Yaskawa INFORM job: X2_7,1(-165,-90)0.JBI

/JOB
//NAME X2_7,1(-165,-90)0
//POS
///NPOS 176,176,176,10,0,0
///TOOL 0
///POSTYPE PULSE
///PULSE
C00000=-39612,-76551,-106625,19964,71626,76894
C00001=-136747,-74177,-105509,19364,71994,77223
C00002=-161484,-91945,-110261,14957,103238,71453
C00003=-134320,-92773,-58904,770,74516,77205
C00004=-134673,-92214,-54444,791,72061,77068
C00005=-134820,-91899,-52604,800,71092,77011
C00006=-134844,-90764,-50356,804,70293,76998
C00007=-134845,-90951,-50699,804,70408,76998
C00008=-134847,-90902,-50689,804,70426,76998
C00009=-135220,-93018,-51550,819,69873,76866
C00010=-134847,-90902,-50689,804,70426,76998
C00011=-134345,-91899,-57067,774,73834,77192
C00012=-131570,-88662,-77507,437,88211,78221
C00013=-134523,-105271,-82138,1688,77555,77123
C00014=-134783,-105110,-77920,1731,75048,76999
C00015=-134891,-104934,-76180,1749,74070,76947
C00016=-134915,-104095,-74155,1758,73257,76927
C00017=-134916,-104246,-74475,1757,73376,76929
C00018=-134967,-104172,-74385,1762,73360,76911
C00019=-135343,-106731,-75345,1806,72644,76769
C00020=-134967,-104172,-74385,1762,73360,76911
C00021=-134596,-104670,-80422,1700,76809,77088
C00022=-136142,-134585,-102052,6475,55790,75677
C00023=-135158,-114824,-94391,5988,60976,76349
C00024=-135004,-111643,-89125,6022,59367,76321
C00025=-134943,-110346,-86998,6037,58724,76309
C00026=-134968,-109685,-85073,6101,57885,76253
C00027=-134968,-109829,-85430,6091,58030,76261
C00028=-135015,-109667,-85346,6108,58065,76244
C00029=-135392,-112540,-86390,6315,57265,76048
C00030=-135015,-109667,-85346,6108,58065,76244
C00031=-135230,-114226,-92783,6055,60303,76285
C00032=-156325,-82511,-105508,20476,72304,69745
C00033=-137289,-84891,-120500,10173,76813,76449
C00034=-137303,-139323,-128947,10263,31295,76421
C00035=-31263,-162610,-128854,9653,11963,76756
C00036=11604,-169116,-125244,11553,23484,75880
C00037=126218,-114256,-117174,36511,17097,65041
C00038=160817,-140540,-109431,13437,75130,4571
C00039=171379,-93893,-58713,11798,67401,-77246
C00040=173134,-92396,-53907,11771,65008,-76852
C00041=173854,-91715,-51934,11761,64060,-76687
C00042=173992,-90510,-49657,11819,63274,-76718
C00043=173854,-91715,-51934,11761,64060,-76687
C00044=173987,-90681,-50014,11807,63403,-76706
C00045=175295,-92334,-50710,11680,62808,-76287
C00046=173987,-90681,-50014,11807,63403,-76706
C00047=173264,-91392,-52007,11815,64350,-76873
C00048=171504,-92964,-56866,11837,66737,-77269
C00049=148375,-121212,-86833,17149,72660,-74878
C00050=158259,-104656,-80103,12690,76821,-80970
C00051=159746,-104467,-75973,12677,74202,-80717
C00052=160359,-104277,-74268,12676,73177,-80607
C00053=160467,-103358,-72208,12716,72383,-80652
C00054=160359,-104277,-74268,12676,73177,-80607
C00055=160417,-103437,-72504,12711,72529,-80655
C00056=161432,-105657,-73351,12654,71766,-80373
C00057=160417,-103437,-72504,12711,72529,-80655
C00058=159802,-103665,-74229,12711,73547,-80766
C00059=158313,-103959,-78409,12718,76144,-81021
C00060=158569,-141300,-112815,9916,80451,-74883
C00061=158798,-111123,-96627,9897,85638,-81727
C00062=159864,-112561,-93144,9862,82666,-81595
C00063=160305,-112963,-91680,9854,81520,-81533
C00064=160413,-112330,-89778,9865,80674,-81563
C00065=160399,-112442,-90081,9863,80802,-81557
C00066=160441,-112453,-90085,9860,80794,-81544
C00067=161459,-115136,-91053,9809,79898,-81262
C00068=160441,-112453,-90085,9860,80794,-81544
C00069=159997,-112112,-91574,9867,81924,-81608
C00070=158926,-110847,-95124,9896,84850,-81745
C00071=160682,-88290,-103875,4722,98055,-77441
C00072=135323,-109589,-91807,-1190,81195,-77099
C00073=133148,-118247,-66270,-328,65792,-77561
C00074=133675,-116428,-61229,-353,63627,-77373
C00075=133898,-115629,-59169,-363,62770,-77293
C00076=133957,-114036,-56802,-368,62133,-77271
C00077=133948,-114328,-57228,-367,62244,-77274
C00078=133917,-114378,-57192,-366,62197,-77284
C00079=134431,-116412,-57765,-387,61506,-77104
C00080=133917,-114378,-57192,-366,62197,-77284
C00081=133693,-115200,-59270,-355,63052,-77365
C00082=133162,-117080,-64355,-330,65213,-77555
C00083=138392,-136781,-94069,-1907,68850,-75598
C00084=132958,-105241,-81767,-1134,77157,-77611
C00085=133235,-105027,-77525,-1173,74661,-77491
C00086=133288,-104357,-75613,-1183,73831,-77465
C00087=133388,-103974,-73743,-1199,72877,-77421
C00088=133382,-104139,-74110,-1197,73019,-77424
C00089=133359,-104157,-74082,-1195,72992,-77432
C00090=133697,-106715,-75039,-1234,72272,-77307
C00091=133359,-104157,-74082,-1195,72992,-77432
C00092=133244,-104394,-75853,-1178,73958,-77481
C00093=132967,-104722,-80150,-1137,76429,-77601
C00094=138196,-141776,-101555,-7752,51920,-74477
C00095=133428,-114968,-94090,-4986,60450,-76927
C00096=133334,-111722,-88803,-5027,58864,-76892
C00097=133296,-110401,-86667,-5046,58229,-76877
C00098=133336,-109716,-84733,-5107,57396,-76822
C00099=133330,-109844,-85063,-5097,57532,-76831
C00100=133345,-109829,-85035,-5104,57524,-76825
C00101=133683,-112700,-86073,-5289,56713,-76650
C00102=133345,-109829,-85035,-5104,57524,-76825
C00103=133382,-111175,-87184,-5084,58155,-76839
C00104=133477,-114487,-92506,-5041,59728,-76875
C00105=141752,-106189,-89524,-13947,62090,-73527
C00106=139337,-93830,-82897,-11067,68844,-75160
C00107=137529,-73575,-73827,-8033,82117,-76735
C00108=128276,-76076,-75002,-6276,80740,-79812
C00109=127910,-97020,-84121,-7469,66652,-79182
C00110=129021,-107399,-90499,-8627,61500,-78401
C00111=153189,-105013,-101528,-11669,72335,-68251
C00112=139010,-107606,-90936,13602,98517,-80019
C00113=140479,-111236,-88693,13669,95112,-79881
C00114=141104,-112370,-87439,13712,93689,-79820
C00115=153388,-106096,-85115,15113,93243,-75565
C00116=152633,-104764,-86492,15083,94863,-75632
C00117=150753,-101320,-88700,15024,98237,-75883
C00118=160913,-92989,-79235,24173,97682,-73194
C00119=151950,-102059,-74371,18707,88669,-80768
C00120=154021,-103736,-71350,18921,85616,-80507
C00121=156769,-103064,-69269,19190,84099,-79774
C00122=166959,-95557,-66660,19849,83821,-76203
C00123=165303,-95872,-68594,19733,85187,-76570
C00124=162983,-94318,-71559,19573,88219,-76909
C00125=177330,-95873,-81273,-5233,90327,-76206
C00126=140937,-97211,-77708,-6493,80278,-75430
C00127=139211,-88421,-70354,-5139,84673,-76249
C00128=139768,-88806,-68107,-5161,83133,-75995
C00129=129086,-91534,-69174,-4923,81722,-79583
C00130=127811,-91239,-71468,-4873,83202,-80077
C00131=128888,-101422,-79212,-5537,77745,-79462
C00132=137877,-110952,-72155,-1851,88703,-77001
C00133=139734,-110509,-58972,-1399,80627,-76317
C00134=140249,-110783,-54995,-1319,78047,-76125
C00135=142549,-109961,-52712,-916,77094,-75392
C00136=133855,-111346,-52444,-6859,76619,-78478
C00137=133337,-111815,-54560,-7332,77679,-78736
C00138=134028,-111541,-58531,-7151,80301,-78669
C00139=164216,-109032,-67322,9813,79557,-67843
C00140=178281,-110359,-72151,20782,77591,-61941
C00141=158557,-96763,-53299,19671,77500,-80212
C00142=161145,-96732,-49400,20091,74655,-79786
C00143=163160,-95939,-47445,20342,73441,-79290
C00144=171236,-91338,-45159,23204,70710,-76469
C00145=169251,-92133,-47198,23012,72018,-76926
C00146=166209,-92508,-51159,22625,74900,-77459
C00147=149807,-144247,-110382,14568,75746,-63630
C00148=126218,-114256,-117174,36511,17097,65041
C00149=118793,-153239,-128782,32477,23422,65112
C00150=11604,-169116,-125244,11553,23484,75880
C00151=-137287,-84892,-120500,10191,64594,76446
C00152=-160620,-101266,-113002,23179,68693,67515
C00153=-142986,-103863,-89383,14232,64402,73407
C00154=-140772,-93459,-83022,11808,69469,74770
C00155=-137440,-81398,-77271,8908,76967,76533
C00156=-127109,-84097,-78453,6470,75327,80029
C00157=-129407,-96992,-84444,8303,67122,78735
C00158=-131023,-111117,-91294,10327,58712,77443
C00159=-137851,-122869,-93518,6619,76408,76346
C00160=-142777,-98750,-78529,7299,79569,74803
C00161=-140556,-88306,-70608,5557,85156,75864
C00162=-139393,-89232,-68583,5550,83361,76182
C00163=-128741,-91750,-69554,5331,81947,79756
C00164=-129199,-91422,-71906,5329,83587,79669
C00165=-130949,-106780,-81238,6593,74219,78605
C00166=-147304,-112155,-77948,4789,93136,74966
C00167=-140707,-86501,-53635,6284,90799,77049
C00168=-140521,-88167,-50612,6312,88084,76975
C00169=-139464,-88632,-48933,6512,86739,77253
C00170=-126799,-90769,-49711,8803,84964,81310
C00171=-127817,-90605,-51563,8619,86280,81066
C00172=-128613,-89112,-54690,8476,89025,80988
C00173=-161484,-91945,-110261,14957,103238,71453
C00174=-136747,-74177,-105509,19364,71994,77223
C00175=-39612,-76551,-106625,19964,71626,76894
BC00000=295325,674563,1075175
BC00001=353535,895977,1075175
BC00002=353535,975867,1075175
BC00003=346138,1016365,1074941
BC00004=346138,1016365,1074941
BC00005=346138,1016365,1074941
BC00006=346138,1016365,1074941
BC00007=346138,1016365,1074941
BC00008=346138,1016365,1074941
BC00009=346138,1016365,1074941
BC00010=346138,1016365,1074941
BC00011=346138,1016365,1074941
BC00012=345633,1015596,1047596
BC00013=345436,1039539,1075175
BC00014=345436,1039539,1075175
BC00015=345436,1039539,1075175
BC00016=345436,1039539,1075175
BC00017=345436,1039539,1075175
BC00018=345436,1039539,1075175
BC00019=345436,1039539,1075175
BC00020=345436,1039539,1075175
BC00021=345436,1039539,1075175
BC00022=345633,1030850,1075175
BC00023=346084,1031619,1075175
BC00024=346084,1031619,1075175
BC00025=346084,1031619,1075175
BC00026=346084,1031619,1075175
BC00027=346084,1031619,1075175
BC00028=346084,1031619,1075175
BC00029=346084,1031619,1075175
BC00030=346084,1031619,1075175
BC00031=346084,1031619,1075175
BC00032=381896,966588,1075175
BC00033=353816,923989,1075175
BC00034=353816,923989,1075175
BC00035=379773,1126391,1075175
BC00036=335955,1030285,1075175
BC00037=312632,1138057,1075175
BC00038=340753,1115300,1075175
BC00039=317618,1085268,1067802
BC00040=317618,1085268,1067802
BC00041=317618,1085268,1067802
BC00042=317618,1085268,1067802
BC00043=317618,1085268,1067802
BC00044=317618,1085268,1067802
BC00045=317618,1085268,1067802
BC00046=317618,1085268,1067802
BC00047=317618,1085268,1067802
BC00048=317618,1085268,1067802
BC00049=304558,1071386,1075175
BC00050=304527,1061353,1075175
BC00051=304527,1061353,1075175
BC00052=304527,1061353,1075175
BC00053=304527,1061353,1075175
BC00054=304527,1061353,1075175
BC00055=304527,1061353,1075175
BC00056=304527,1061353,1075175
BC00057=304527,1061353,1075175
BC00058=304527,1061353,1075175
BC00059=304527,1061353,1075175
BC00060=297809,1030861,1075175
BC00061=297809,1030861,1075175
BC00062=297809,1030861,1075175
BC00063=297809,1030861,1075175
BC00064=297809,1030861,1075175
BC00065=297809,1030861,1075175
BC00066=297809,1030861,1075175
BC00067=297809,1030861,1075175
BC00068=297809,1030861,1075175
BC00069=297809,1030861,1075175
BC00070=297809,1030861,1075175
BC00071=323405,1100688,1075175
BC00072=345633,1145987,1075175
BC00073=341431,1080783,1075175
BC00074=341431,1080783,1075175
BC00075=341431,1080783,1075175
BC00076=341431,1080783,1075175
BC00077=341431,1080783,1075175
BC00078=341431,1080783,1075175
BC00079=341431,1080783,1075175
BC00080=341431,1080783,1075175
BC00081=341431,1080783,1075175
BC00082=341431,1080783,1075175
BC00083=345633,1085057,1075175
BC00084=345596,1084288,1075175
BC00085=345596,1084288,1075175
BC00086=345596,1084288,1075175
BC00087=345596,1084288,1075175
BC00088=345596,1084288,1075175
BC00089=345596,1084288,1075175
BC00090=345596,1084288,1075175
BC00091=345596,1084288,1075175
BC00092=345596,1084288,1075175
BC00093=345596,1084288,1075175
BC00094=345633,1092894,1075175
BC00095=345573,1092125,1075175
BC00096=345573,1092125,1075175
BC00097=345573,1092125,1075175
BC00098=345573,1092125,1075175
BC00099=345573,1092125,1075175
BC00100=345573,1092125,1075175
BC00101=345573,1092125,1075175
BC00102=345573,1092125,1075175
BC00103=345573,1092125,1075175
BC00104=345573,1092125,1075175
BC00105=338421,1101651,1075175
BC00106=338421,1101651,1075175
BC00107=338421,1101651,1075175
BC00108=338421,1101651,1075175
BC00109=338421,1101651,1075175
BC00110=338421,1101651,1075175
BC00111=329561,1092894,1075175
BC00112=285121,1016140,1075175
BC00113=285121,1016140,1075175
BC00114=285121,1016140,1075175
BC00115=285121,1016140,1075175
BC00116=285121,1016140,1075175
BC00117=285121,1016140,1075175
BC00118=322883,1030260,1075175
BC00119=305317,1037338,1075175
BC00120=305317,1037338,1075175
BC00121=305317,1037338,1075175
BC00122=305317,1037338,1075175
BC00123=305317,1037338,1075175
BC00124=305317,1037338,1075175
BC00125=352461,1065435,1075175
BC00126=338520,1089250,1075175
BC00127=338520,1089250,1075175
BC00128=338520,1089250,1075175
BC00129=338520,1089250,1075175
BC00130=338520,1089250,1075175
BC00131=338520,1089250,1075175
BC00132=329561,1063988,1075175
BC00133=329824,1054944,1075175
BC00134=329824,1054944,1075175
BC00135=329824,1054944,1075175
BC00136=329824,1054944,1075175
BC00137=329824,1054944,1075175
BC00138=329824,1054944,1075175
BC00139=331300,1058024,1069499
BC00140=329561,1042367,1075175
BC00141=308437,1059196,1075175
BC00142=308437,1059196,1075175
BC00143=308437,1059196,1075175
BC00144=308437,1059196,1075175
BC00145=308437,1059196,1075175
BC00146=308437,1059196,1075175
BC00147=340753,1115300,1075175
BC00148=312632,1138057,1075175
BC00149=312632,1138057,1075175
BC00150=335955,1030285,1075175
BC00151=353817,923990,1075175
BC00152=381896,966588,1075175
BC00153=338906,1022094,1075175
BC00154=338906,1022094,1075175
BC00155=338906,1022094,1075175
BC00156=338906,1022094,1075175
BC00157=338906,1022094,1075175
BC00158=338906,1022094,1075175
BC00159=330026,1050278,1075175
BC00160=338884,1034595,1075175
BC00161=338884,1034595,1075175
BC00162=338884,1034595,1075175
BC00163=338884,1034595,1075175
BC00164=338884,1034595,1075175
BC00165=338884,1034595,1075175
BC00166=330026,1059203,1075175
BC00167=326517,1040873,1058771
BC00168=326517,1040873,1058771
BC00169=326517,1040873,1058771
BC00170=326517,1040873,1058771
BC00171=326517,1040873,1058771
BC00172=326517,1040873,1058771
BC00173=353535,975867,1075175
BC00174=353535,895977,1075175
BC00175=295325,674563,1075175
EC00000=-1463287,-556475
EC00001=-1463287,-556475
EC00002=-1463287,-556475
EC00003=-1463287,-556475
EC00004=-1463287,-556475
EC00005=-1463287,-556475
EC00006=-1463287,-556475
EC00007=-1463287,-556475
EC00008=-1463287,-556475
EC00009=-1463287,-556475
EC00010=-1463287,-556475
EC00011=-1463287,-556475
EC00012=-1463287,-556475
EC00013=-1463287,-556475
EC00014=-1463287,-556475
EC00015=-1463287,-556475
EC00016=-1463287,-556475
EC00017=-1463287,-556475
EC00018=-1463287,-556475
EC00019=-1463287,-556475
EC00020=-1463287,-556475
EC00021=-1463287,-556475
EC00022=-1463287,-556475
EC00023=-1463287,-556475
EC00024=-1463287,-556475
EC00025=-1463287,-556475
EC00026=-1463287,-556475
EC00027=-1463287,-556475
EC00028=-1463287,-556475
EC00029=-1463287,-556475
EC00030=-1463287,-556475
EC00031=-1463287,-556475
EC00032=-1463287,-556475
EC00033=-1463287,-556475
EC00034=-1463287,-556475
EC00035=-1463287,-556475
EC00036=-1595090,-3837
EC00037=-1729339,556475
EC00038=-1729339,556475
EC00039=-1729339,556475
EC00040=-1729339,556475
EC00041=-1729339,556475
EC00042=-1729339,556475
EC00043=-1729339,556475
EC00044=-1729339,556475
EC00045=-1729339,556475
EC00046=-1729339,556475
EC00047=-1729339,556475
EC00048=-1729339,556475
EC00049=-1729339,556475
EC00050=-1729339,556475
EC00051=-1729339,556475
EC00052=-1729339,556475
EC00053=-1729339,556475
EC00054=-1729339,556475
EC00055=-1729339,556475
EC00056=-1729339,556475
EC00057=-1729339,556475
EC00058=-1729339,556475
EC00059=-1729339,556475
EC00060=-1729339,556475
EC00061=-1729339,556475
EC00062=-1729339,556475
EC00063=-1729339,556475
EC00064=-1729339,556475
EC00065=-1729339,556475
EC00066=-1729339,556475
EC00067=-1729339,556475
EC00068=-1729339,556475
EC00069=-1729339,556475
EC00070=-1729339,556475
EC00071=-1729339,556475
EC00072=-1729339,556475
EC00073=-1729339,556475
EC00074=-1729339,556475
EC00075=-1729339,556475
EC00076=-1729339,556475
EC00077=-1729339,556475
EC00078=-1729339,556475
EC00079=-1729339,556475
EC00080=-1729339,556475
EC00081=-1729339,556475
EC00082=-1729339,556475
EC00083=-1729339,556475
EC00084=-1729339,556475
EC00085=-1729339,556475
EC00086=-1729339,556475
EC00087=-1729339,556475
EC00088=-1729339,556475
EC00089=-1729339,556475
EC00090=-1729339,556475
EC00091=-1729339,556475
EC00092=-1729339,556475
EC00093=-1729339,556475
EC00094=-1729339,556475
EC00095=-1729339,556475
EC00096=-1729339,556475
EC00097=-1729339,556475
EC00098=-1729339,556475
EC00099=-1729339,556475
EC00100=-1729339,556475
EC00101=-1729339,556475
EC00102=-1729339,556475
EC00103=-1729339,556475
EC00104=-1729339,556475
EC00105=-1729339,556475
EC00106=-1729339,556475
EC00107=-1729339,556475
EC00108=-1729339,556475
EC00109=-1729339,556475
EC00110=-1729339,556475
EC00111=-1729339,556475
EC00112=-1729339,556475
EC00113=-1729339,556475
EC00114=-1729339,556475
EC00115=-1729339,556475
EC00116=-1729339,556475
EC00117=-1729339,556475
EC00118=-1729339,556475
EC00119=-1729339,556475
EC00120=-1729339,556475
EC00121=-1729339,556475
EC00122=-1729339,556475
EC00123=-1729339,556475
EC00124=-1729339,556475
EC00125=-1729339,556475
EC00126=-1729339,556475
EC00127=-1729339,556475
EC00128=-1729339,556475
EC00129=-1729339,556475
EC00130=-1729339,556475
EC00131=-1729339,556475
EC00132=-1729339,556475
EC00133=-1729339,556475
EC00134=-1729339,556475
EC00135=-1729339,556475
EC00136=-1729339,556475
EC00137=-1729339,556475
EC00138=-1729339,556475
EC00139=-1729339,556475
EC00140=-1729339,556475
EC00141=-1729339,556475
EC00142=-1729339,556475
EC00143=-1729339,556475
EC00144=-1729339,556475
EC00145=-1729339,556475
EC00146=-1729339,556475
EC00147=-1729339,556475
EC00148=-1729339,556475
EC00149=-1729339,556475
EC00150=-1595090,-3837
EC00151=-1463287,-556475
EC00152=-1463287,-556475
EC00153=-1463287,-556475
EC00154=-1463287,-556475
EC00155=-1463287,-556475
EC00156=-1463287,-556475
EC00157=-1463287,-556475
EC00158=-1463287,-556475
EC00159=-1463287,-556475
EC00160=-1463287,-556475
EC00161=-1463287,-556475
EC00162=-1463287,-556475
EC00163=-1463287,-556475
EC00164=-1463287,-556475
EC00165=-1463287,-556475
EC00166=-1463287,-556475
EC00167=-1463287,-556475
EC00168=-1463287,-556475
EC00169=-1463287,-556475
EC00170=-1463287,-556475
EC00171=-1463287,-556475
EC00172=-1463287,-556475
EC00173=-1463287,-556475
EC00174=-1463287,-556475
EC00175=-1463287,-556475
///POSTYPE BASE
///RECTAN
///RCONF 0,0,0,0,0,0,0,0,0,0,0,0,0,0,0,0,0,0,0,0,0,0,0,0
P00006=0.222,-3.123,-1.508,0.0000,0.0000,0.0000
P00021=-0.225,-6.128,-0.405,0.0000,0.0000,0.0000
P00022=0.222,-3.123,-1.508,0.0000,0.0000,0.0000
P00023=0.143,-0.036,0.682,0.0000,0.0000,0.0000
P00031=1.853,-0.001,-1.549,0.0000,0.0000,0.0000
P00032=1.957,0.503,-7.217,0.0000,0.0000,0.0000
///RCONF 0,0,0,0,1,0,0,0,0,0,0,0,0,0,0,0,0,0,0,0,0,0,0,0
P00033=-0.123,0.612,-5.012,0.0000,0.0000,0.0000
///RCONF 0,0,0,0,0,0,0,0,0,0,0,0,0,0,0,0,0,0,0,0,0,0,0,0
P00034=-0.304,0.773,-2.693,0.0000,0.0000,0.0000
P00035=2.817,0.591,-1.622,0.0000,0.0000,0.0000
P00036=-1.108,-0.829,1.850,0.0000,0.0000,0.0000
//INST
///DATE 2024/04/10 10:51
///ATTR SC,RW
///GROUP1 RB1,BS1
///GROUP2 ST1
NOP
'X2_7,1(-165,-90)0
MOVJ C00000 BC00000 VJ=100.00  +MOVJ EC00000 VJ=100.00
MOVJ C00001 BC00001 VJ=100.00  +MOVJ EC00001 VJ=100.00
MOVJ C00002 BC00002 VJ=100.00  +MOVJ EC00002 VJ=100.00
'Path S3195
SFTOF3D
MOVJ C00003 BC00003 VJ=100.00  +MOVJ EC00003 VJ=100.00
MOVL C00004 BC00004 V=800.0  +MOVJ EC00004 VJ=100.00
SMOVL C00005 BC00005 V=166.7  +MOVJ EC00005
SREFP 3 C00006 BC00006  +REFP EC00006
CALL JOB:SEARCH-R1-S13D
SET P021 P006
SFTON3D P021
SMOVL C00007 BC00007 V=166.7  +MOVJ EC00007
SMOVL C00008 BC00008 V=166.7  +MOVJ EC00008
SREFP 3 C00009 BC00009  +REFP EC00009
CALL JOB:SEARCH-R1-S13D
SET P021 P006
SFTON3D P021
SMOVL C00010 BC00010 V=166.7  +MOVJ EC00010
MOVL C00011 BC00011 V=1000.0  +MOVJ EC00011 VJ=100.00
'EndPath S3195
MOVJ C00012 BC00012 VJ=100.00  +MOVJ EC00012 VJ=100.00
'Path S3196
SFTOF3D
MOVJ C00013 BC00013 VJ=100.00  +MOVJ EC00013 VJ=100.00
MOVL C00014 BC00014 V=800.0  +MOVJ EC00014 VJ=100.00
SMOVL C00015 BC00015 V=166.7  +MOVJ EC00015
SREFP 3 C00016 BC00016  +REFP EC00016
CALL JOB:SEARCH-R1-S13D
SET P022 P006
SFTON3D P022
SMOVL C00017 BC00017 V=166.7  +MOVJ EC00017
SMOVL C00018 BC00018 V=166.7  +MOVJ EC00018
SREFP 3 C00019 BC00019  +REFP EC00019
CALL JOB:SEARCH-R1-S13D
SET P022 P006
SFTON3D P022
SMOVL C00020 BC00020 V=166.7  +MOVJ EC00020
MOVL C00021 BC00021 V=1000.0  +MOVJ EC00021 VJ=100.00
'EndPath S3196
MOVJ C00022 BC00022 VJ=100.00  +MOVJ EC00022 VJ=100.00
'Path S3197
SFTOF3D
MOVJ C00023 BC00023 VJ=100.00  +MOVJ EC00023 VJ=100.00
MOVL C00024 BC00024 V=800.0  +MOVJ EC00024 VJ=100.00
SMOVL C00025 BC00025 V=166.7  +MOVJ EC00025
SREFP 3 C00026 BC00026  +REFP EC00026
CALL JOB:SEARCH-R1-S13D
SET P023 P006
SFTON3D P023
SMOVL C00027 BC00027 V=166.7  +MOVJ EC00027
SMOVL C00028 BC00028 V=166.7  +MOVJ EC00028
SREFP 3 C00029 BC00029  +REFP EC00029
CALL JOB:SEARCH-R1-S13D
SET P023 P006
SFTON3D P023
SMOVL C00030 BC00030 V=166.7  +MOVJ EC00030
MOVL C00031 BC00031 V=1000.0  +MOVJ EC00031 VJ=100.00
'EndPath S3197
'obrot
MOVJ C00032 BC00032 VJ=100.00  +MOVJ EC00032 VJ=100.00
MOVJ C00033 BC00033 VJ=100.00  +MOVJ EC00033 VJ=100.00
MOVJ C00034 BC00034 VJ=100.00  +MOVJ EC00034 VJ=100.00
MOVJ C00035 BC00035 VJ=100.00  +MOVJ EC00035 VJ=100.00
MOVJ C00036 BC00036 VJ=100.00  +MOVJ EC00036 VJ=100.00
MOVJ C00037 BC00037 VJ=100.00  +MOVJ EC00037 VJ=100.00
MOVJ C00038 BC00038 VJ=100.00  +MOVJ EC00038 VJ=100.00
'
'Path S3198
SFTOF3D
MOVJ C00039 BC00039 VJ=100.00  +MOVJ EC00039 VJ=100.00
MOVL C00040 BC00040 V=800.0  +MOVJ EC00040 VJ=100.00
SMOVL C00041 BC00041 V=166.7  +MOVJ EC00041
SREFP 3 C00042 BC00042  +REFP EC00042
CALL JOB:SEARCH-R1-S13D
SET P031 P006
SFTON3D P031
SMOVL C00043 BC00043 V=166.7  +MOVJ EC00043
SMOVL C00044 BC00044 V=166.7  +MOVJ EC00044
SREFP 3 C00045 BC00045  +REFP EC00045
CALL JOB:SEARCH-R1-S13D
SET P031 P006
SFTON3D P031
SMOVL C00046 BC00046 V=166.7  +MOVJ EC00046
MOVL C00047 BC00047 V=800.0  +MOVJ EC00047 VJ=100.00
MOVL C00048 BC00048 V=1000.0  +MOVJ EC00048 VJ=100.00
'EndPath S3198
MOVJ C00049 BC00049 VJ=100.00  +MOVJ EC00049 VJ=100.00
'Path S3199
SFTOF3D
MOVJ C00050 BC00050 VJ=100.00  +MOVJ EC00050 VJ=100.00
MOVL C00051 BC00051 V=800.0  +MOVJ EC00051 VJ=100.00
SMOVL C00052 BC00052 V=166.7  +MOVJ EC00052
SREFP 3 C00053 BC00053  +REFP EC00053
CALL JOB:SEARCH-R1-S13D
SET P032 P006
SFTON3D P032
SMOVL C00054 BC00054 V=166.7  +MOVJ EC00054
SMOVL C00055 BC00055 V=166.7  +MOVJ EC00055
SREFP 3 C00056 BC00056  +REFP EC00056
CALL JOB:SEARCH-R1-S13D
SET P032 P006
SFTON3D P032
SMOVL C00057 BC00057 V=166.7  +MOVJ EC00057
MOVL C00058 BC00058 V=800.0  +MOVJ EC00058 VJ=100.00
MOVL C00059 BC00059 V=1000.0  +MOVJ EC00059 VJ=100.00
'EndPath S3199
MOVJ C00060 BC00060 VJ=100.00  +MOVJ EC00060 VJ=100.00
'Path S3200
SFTOF3D
MOVJ C00061 BC00061 VJ=100.00  +MOVJ EC00061 VJ=100.00
MOVL C00062 BC00062 V=800.0  +MOVJ EC00062 VJ=100.00
SMOVL C00063 BC00063 V=166.7  +MOVJ EC00063
SREFP 3 C00064 BC00064  +REFP EC00064
CALL JOB:SEARCH-R1-S13D
SET P033 P006
SFTON3D P033
SMOVL C00065 BC00065 V=166.7  +MOVJ EC00065
SMOVL C00066 BC00066 V=166.7  +MOVJ EC00066
SREFP 3 C00067 BC00067  +REFP EC00067
CALL JOB:SEARCH-R1-S13D
SET P033 P006
SFTON3D P033
SMOVL C00068 BC00068 V=166.7  +MOVJ EC00068
MOVL C00069 BC00069 V=800.0  +MOVJ EC00069 VJ=100.00
MOVL C00070 BC00070 V=1000.0  +MOVJ EC00070 VJ=100.00
'EndPath S3200
MOVJ C00071 BC00071 VJ=100.00  +MOVJ EC00071 VJ=100.00
MOVJ C00072 BC00072 VJ=100.00  +MOVJ EC00072 VJ=100.00
'Path S3201
SFTOF3D
MOVJ C00073 BC00073 VJ=100.00  +MOVJ EC00073 VJ=100.00
MOVL C00074 BC00074 V=800.0  +MOVJ EC00074 VJ=100.00
SMOVL C00075 BC00075 V=166.7  +MOVJ EC00075
SREFP 3 C00076 BC00076  +REFP EC00076
CALL JOB:SEARCH-R1-S13D
SET P034 P006
SFTON3D P034
SMOVL C00077 BC00077 V=166.7  +MOVJ EC00077
SMOVL C00078 BC00078 V=166.7  +MOVJ EC00078
SREFP 3 C00079 BC00079  +REFP EC00079
CALL JOB:SEARCH-R1-S13D
SET P034 P006
SFTON3D P034
SMOVL C00080 BC00080 V=166.7  +MOVJ EC00080
MOVL C00081 BC00081 V=800.0  +MOVJ EC00081 VJ=100.00
MOVL C00082 BC00082 V=1000.0  +MOVJ EC00082 VJ=100.00
'EndPath S3201
MOVJ C00083 BC00083 VJ=100.00  +MOVJ EC00083 VJ=100.00
'Path S3202
SFTOF3D
MOVJ C00084 BC00084 VJ=100.00  +MOVJ EC00084 VJ=100.00
MOVL C00085 BC00085 V=800.0  +MOVJ EC00085 VJ=100.00
SMOVL C00086 BC00086 V=166.7  +MOVJ EC00086
SREFP 3 C00087 BC00087  +REFP EC00087
CALL JOB:SEARCH-R1-S13D
SET P035 P006
SFTON3D P035
SMOVL C00088 BC00088 V=166.7  +MOVJ EC00088
SMOVL C00089 BC00089 V=166.7  +MOVJ EC00089
SREFP 3 C00090 BC00090  +REFP EC00090
CALL JOB:SEARCH-R1-S13D
SET P035 P006
SFTON3D P035
SMOVL C00091 BC00091 V=166.7  +MOVJ EC00091
MOVL C00092 BC00092 V=800.0  +MOVJ EC00092 VJ=100.00
MOVL C00093 BC00093 V=1000.0  +MOVJ EC00093 VJ=100.00
'EndPath S3202
MOVJ C00094 BC00094 VJ=100.00  +MOVJ EC00094 VJ=100.00
'Path S3203
SFTOF3D
MOVJ C00095 BC00095 VJ=100.00  +MOVJ EC00095 VJ=100.00
MOVL C00096 BC00096 V=800.0  +MOVJ EC00096 VJ=100.00
SMOVL C00097 BC00097 V=166.7  +MOVJ EC00097
SREFP 3 C00098 BC00098  +REFP EC00098
CALL JOB:SEARCH-R1-S13D
SET P036 P006
SFTON3D P036
SMOVL C00099 BC00099 V=166.7  +MOVJ EC00099
SMOVL C00100 BC00100 V=166.7  +MOVJ EC00100
SREFP 3 C00101 BC00101  +REFP EC00101
CALL JOB:SEARCH-R1-S13D
SET P036 P006
SFTON3D P036
SMOVL C00102 BC00102 V=166.7  +MOVJ EC00102
MOVL C00103 BC00103 V=800.0  +MOVJ EC00103 VJ=100.00
MOVL C00104 BC00104 V=1000.0  +MOVJ EC00104 VJ=100.00
'EndPath S3203
'Path W3204
SFTOF3D
SFTON3D P036
MOVJ C00105 BC00105 VJ=100.00  +MOVJ EC00105 VJ=100.00
SMOVL C00106 BC00106 V=800.0  +MOVJ EC00106
'POSPAWANE 2 SPOINY
SMOVL C00107 BC00107 V=166.7 PL=0  +MOVJ EC00107
MACRO1 MJ#(0) ARGF21
ARCON
SMOVL C00108 BC00108 V=11.7  +MOVJ EC00108
ARCOF
SMOVL C00109 BC00109 V=800.0  +MOVJ EC00109
SMOVL C00110 BC00110 V=1000.0  +MOVJ EC00110
SFTOF3D
'EndPath W3204
MOVJ C00111 BC00111 VJ=100.00  +MOVJ EC00111 VJ=100.00
'Path W3205
SFTOF3D
SFTON3D P033
MOVJ C00112 BC00112 VJ=100.00  +MOVJ EC00112 VJ=100.00
SMOVL C00113 BC00113 V=800.0  +MOVJ EC00113
SMOVL C00114 BC00114 V=166.7 PL=0  +MOVJ EC00114
ARCON
SMOVL C00115 BC00115 V=11.7  +MOVJ EC00115
ARCOF
SMOVL C00116 BC00116 V=800.0  +MOVJ EC00116
SMOVL C00117 BC00117 V=1000.0  +MOVJ EC00117
SFTOF3D
'EndPath W3205
MOVJ C00118 BC00118 VJ=100.00  +MOVJ EC00118 VJ=100.00
'Path W3206
SFTOF3D
SFTON3D P032
MOVJ C00119 BC00119 VJ=100.00  +MOVJ EC00119 VJ=100.00
SMOVL C00120 BC00120 V=800.0  +MOVJ EC00120
SMOVL C00121 BC00121 V=166.7 PL=0  +MOVJ EC00121
MACRO1 MJ#(0) ARGF14
ARCON
SMOVL C00122 BC00122 V=11.7  +MOVJ EC00122
ARCOF
SMOVL C00123 BC00123 V=800.0  +MOVJ EC00123
SMOVL C00124 BC00124 V=1000.0  +MOVJ EC00124
SFTOF3D
'EndPath W3206
MOVJ C00125 BC00125 VJ=100.00  +MOVJ EC00125 VJ=100.00
'Path W3207
SFTOF3D
SFTON3D P035
MOVJ C00126 BC00126 VJ=100.00  +MOVJ EC00126 VJ=100.00
SMOVL C00127 BC00127 V=800.0  +MOVJ EC00127
SMOVL C00128 BC00128 V=166.7 PL=0  +MOVJ EC00128
ARCON
SMOVL C00129 BC00129 V=11.7  +MOVJ EC00129
ARCOF
SMOVL C00130 BC00130 V=800.0  +MOVJ EC00130
SMOVL C00131 BC00131 V=1000.0  +MOVJ EC00131
SFTOF3D
'EndPath W3207
MOVJ C00132 BC00132 VJ=100.00  +MOVJ EC00132 VJ=100.00
'Path W3208
SFTOF3D
SFTON3D P034
MOVJ C00133 BC00133 VJ=100.00  +MOVJ EC00133 VJ=100.00
SMOVL C00134 BC00134 V=800.0  +MOVJ EC00134
SMOVL C00135 BC00135 V=166.7 PL=0  +MOVJ EC00135
ARCON
SMOVL C00136 BC00136 V=11.7  +MOVJ EC00136
ARCOF
SMOVL C00137 BC00137 V=800.0  +MOVJ EC00137
SMOVL C00138 BC00138 V=1000.0  +MOVJ EC00138
SFTOF3D
'EndPath W3208
MOVJ C00139 BC00139 VJ=100.00  +MOVJ EC00139 VJ=100.00
MOVJ C00140 BC00140 VJ=100.00  +MOVJ EC00140 VJ=100.00
'Path W3209
SFTOF3D
SFTON3D P031
MOVJ C00141 BC00141 VJ=100.00  +MOVJ EC00141 VJ=100.00
SMOVL C00142 BC00142 V=800.0  +MOVJ EC00142
SMOVL C00143 BC00143 V=166.7 PL=0  +MOVJ EC00143
ARCON
SMOVL C00144 BC00144 V=11.7  +MOVJ EC00144
ARCOF
SMOVL C00145 BC00145 V=800.0  +MOVJ EC00145
SMOVL C00146 BC00146 V=1000.0  +MOVJ EC00146
SFTOF3D
'EndPath W3209
'obrot
MOVJ C00147 BC00147 VJ=100.00  +MOVJ EC00147 VJ=100.00
MOVJ C00148 BC00148 VJ=100.00  +MOVJ EC00148 VJ=100.00
MOVJ C00149 BC00149 VJ=100.00  +MOVJ EC00149 VJ=100.00
MOVJ C00150 BC00150 VJ=100.00  +MOVJ EC00150 VJ=100.00
MOVJ C00151 BC00151 VJ=100.00  +MOVJ EC00151 VJ=100.00
MOVJ C00152 BC00152 VJ=100.00  +MOVJ EC00152 VJ=100.00
'
'Path W3210
SFTOF3D
SFTON3D P023
MOVJ C00153 BC00153 VJ=100.00  +MOVJ EC00153 VJ=100.00
SMOVL C00154 BC00154 V=800.0  +MOVJ EC00154
SMOVL C00155 BC00155 V=166.7 PL=0  +MOVJ EC00155
ARCON
SMOVL C00156 BC00156 V=11.7  +MOVJ EC00156
ARCOF
SMOVL C00157 BC00157 V=800.0  +MOVJ EC00157
SMOVL C00158 BC00158 V=1000.0  +MOVJ EC00158
SFTOF3D
'EndPath W3210
MOVJ C00159 BC00159 VJ=100.00  +MOVJ EC00159 VJ=100.00
'Path W3211
SFTOF3D
SFTON3D P022
MOVJ C00160 BC00160 VJ=100.00  +MOVJ EC00160 VJ=100.00
SMOVL C00161 BC00161 V=800.0  +MOVJ EC00161
SMOVL C00162 BC00162 V=166.7 PL=0  +MOVJ EC00162
ARCON
SMOVL C00163 BC00163 V=11.7  +MOVJ EC00163
ARCOF
SMOVL C00164 BC00164 V=800.0  +MOVJ EC00164
SMOVL C00165 BC00165 V=1000.0  +MOVJ EC00165
SFTOF3D
'EndPath W3211
MOVJ C00166 BC00166 VJ=100.00  +MOVJ EC00166 VJ=100.00
'Path W3212
SFTOF3D
SFTON3D P021
MOVJ C00167 BC00167 VJ=100.00  +MOVJ EC00167 VJ=100.00
SMOVL C00168 BC00168 V=800.0  +MOVJ EC00168
SMOVL C00169 BC00169 V=166.7 PL=0  +MOVJ EC00169
ARCON
SMOVL C00170 BC00170 V=11.7  +MOVJ EC00170
ARCOF
SMOVL C00171 BC00171 V=800.0  +MOVJ EC00171
SMOVL C00172 BC00172 V=1000.0  +MOVJ EC00172
SFTOF3D
'EndPath W3212
MOVJ C00173 BC00173 VJ=100.00  +MOVJ EC00173 VJ=100.00
MOVJ C00174 BC00174 VJ=100.00  +MOVJ EC00174 VJ=100.00
MOVJ C00175 BC00175 VJ=100.00  +MOVJ EC00175 VJ=100.00
END
